(* IEC 61131-3 sources: ATCMcontrol_Engineering/src/Target/ATHW119/Libs/ATCM_System, 14 files *)

(* ---- _ThrowException.st ---- *)
(*[[
    UserURL= "ATCMfile:ThrowException.htm"
]]*)
(*
 *  ATCMControl Standard Function ThrowException
 *  Purpose: Throws an user exception for the calling task.
 *           NOTE: The task is stopped after the exception.
 *)
FUNCTION _ThrowException

inline{STDLIB(_ThrowException)}

END_FUNCTION

(* ---- ClearLocalTaskErrno.st ---- *)
(*[[
    UserURL= "ATCMfile:ClearLocalTaskErrno.htm"
]]*)
(*
 *  ATCMControl Standard Function ClearLocalTaskErrno
 *  Purpose: Clears the error state of the given task.
 *)
FUNCTION ClearLocalTaskErrno
VAR_INPUT
    NAME : ANY_STRING;
END_VAR

overload (STRING)  inline{STDLIB(ClearLocalTaskErrno)}

END_FUNCTION

(* ---- ClearTaskErrno.st ---- *)
(*[[
    UserURL= "ATCMfile:ClearTaskErrno.htm"
]]*)
(*
 *  ATCMControl Standard Function ClearTaskErrno
 *  Purpose: Clears the error state variable of the
 *           calling task. Error numbers <>0 signal an
 *           error.
 *)
FUNCTION ClearTaskErrno

inline{STDLIB(ClearTaskErrno)}

END_FUNCTION

(* ---- EnableWatchdog.st ---- *)
(*[[
    UserURL= "ATCMfile:EnableWatchdog.htm"
]]*)
(*
 *  ATCMControl Standard Function EnableWatchdog
 *)
FUNCTION EnableWatchdog

VAR_INPUT
    ENABLE : BOOL;
END_VAR

inline{STDLIB(EnableWatchdog)}

END_FUNCTION

(* ---- GetLocalTaskErrno.st ---- *)
(*[[
    UserURL= "ATCMfile:GetLocalTaskErrno.htm"
]]*)
(*
 *  ATCMControl Standard Function GetLocalTaskErrno
 *  Purpose: get the task error number of the named task.
 *           NOTE: name must be given in "lower case".
 *           Return values <>0 signal an error.
 *           See also the FC_ERRNO_* values
 *           defined in ATCM_System.cst.
 *)
FUNCTION GetLocalTaskErrno : DINT
VAR_INPUT
    NAME : ANY_STRING;
END_VAR

overload DINT(STRING)  inline {STDLIB(GetLocalTaskErrno)}

END_FUNCTION

(* ---- GetLocalTaskInfo.st ---- *)
(*[[
    UserURL= "ATCMfile:GetLocalTaskInfo.htm"
]]*)
(*
 *  ATCMControl Standard Function GetLocalTaskInfo
 *)
FUNCTION GetLocalTaskInfo
VAR_INPUT
    NAME : ANY_STRING;
END_VAR

VAR_IN_OUT
    INFO : TASKINFO;
END_VAR

overload (STRING,TASKINFO)  inline{STDLIB(GetLocalTaskInfo)}

END_FUNCTION

(* ---- GetLocalTaskState.st ---- *)
(*[[
    UserURL= "ATCMfile:GetLocalTaskState.htm"
]]*)
(*
 *  ATCMControl Standard Function GetLocalTaskState
 *  Purpose: get the current task execution state of the named task.
 *           NOTE: name must be given in "lower case".
 *  possible return values are (see system.cst):
 * CONST
 *   FC_TASK_STATE_ERROR       : DINT :=-1;
 *   FC_TASK_STATE_ONCREATION  : DINT := 0;
 *   FC_TASK_STATE_STOPPED     : DINT := 1;
 *   FC_TASK_STATE_RUNNING     : DINT := 2;
 *   FC_TASK_STATE_BREAK       : DINT := 3;
 * END_CONST
 *)
FUNCTION GetLocalTaskState : DINT
VAR_INPUT
    NAME : ANY_STRING;
END_VAR

overload DINT(STRING)  inline{STDLIB(GetLocalTaskState)}

END_FUNCTION

(* ---- GetTaskErrno.st ---- *)
(*[[
    UserURL= "ATCMfile:GetTaskErrno.htm"
]]*)
(*
 *  ATCMControl Standard Function GetTaskErrno
 *  Purpose: returns the last error number of the
 *           calling task.
 *           Return values <>0 signal an error.
 *           See also the FC_ERRNO_* values
 *           defined in ATCM_System.cst.
 *)
FUNCTION GetTaskErrno : DINT

inline{STDLIB(GetTaskErrno)}

END_FUNCTION

(* ---- getTimeSinceSystemBoot.st ---- *)
(*[[
    UserURL= "ATCMfile:getTimeSinceSystemBoot.htm"
]]*)

FUNCTION getTimeSinceSystemBoot : TIME

inline{STDLIB(GetTimeSinceSystemBoot)}

END_FUNCTION

(* ---- OutputDebugString.st ---- *)
(*[[
    UserURL= "ATCMfile:OutputDebugString.htm"
]]*)
(*
 *  ATCMControl Standard Functionblock OutputDebugString
 *  Purpose: Write a string to the control's standard output
 *           and the log file. A new line character is added
 *           automatically.
 *)
FUNCTION OutputDebugString
VAR_INPUT
    STR        : ANY_STRING;     (* a one-line message to the user*)
END_VAR

overload (STRING) inline{STDLIB(OutputDebugString)}

END_FUNCTION

(* ---- SFCResetToInitialStep.st ---- *)
(*[[
    UserURL= "ATCMfile:SFCResetToInitialStep.htm"
]]*)
(*
 *  ATCMControl Standard Function SFCResetToInitialStep
 *  Purpose: reset SFC logic
 *)
FUNCTION SFCResetToInitialStep

VAR_INPUT
    ENABLE : BOOL; (* reset only if ENABLE = TRUE *)
END_VAR

inline
{
    push1     %1
    POPD_IN_1    __resetSFC
}

END_FUNCTION

(* ---- StartLocalTask.st ---- *)
(*[[
    UserURL= "ATCMfile:StartLocalTask.htm"
]]*)
(*
 *  ATCMControl Standard Function StartLocalTask
 *  Purpose: Put the named task to the running state.
 *           NOTE: name must be given in "lower case".
 *)
FUNCTION StartLocalTask
VAR_INPUT
    NAME : ANY_STRING;
END_VAR

overload (STRING)  inline{STDLIB(StartLocalTask)}

END_FUNCTION

(* ---- StopLocalTask.st ---- *)
(*[[
    UserURL= "ATCMfile:StopLocalTask.htm"
]]*)
(*
 *  ATCMControl Standard Function StopLocalTask
 *  Purpose: Put the named task to the stopped state.
 *           NOTE: name must be given in "lower case".
 *  WARNING: never try to stop the own task.
 *)
FUNCTION StopLocalTask
VAR_INPUT
    NAME : ANY_STRING;
END_VAR

overload (STRING)  inline{STDLIB(StopLocalTask)}

END_FUNCTION

(* ---- SignalError.st ---- *)
(*[[
    UserURL= "ATCMfile:SignalError.htm"
]]*)
(*
 *  ATCMControl Standard Functionblock SignalError
 *  Purpose: Send Task to Error State
 *
 *  if enable=TRUE and errno<>0 then
 *    the current task is stopped.
 *)
FUNCTION_BLOCK SignalError

VAR_INPUT
    ENABLE     : BOOL:=TRUE;  (* enable this inst *)
    ERRNO      : DINT:=0;     (* error number *)
END_VAR

inline{STDLIB(SignalError)}

END_FUNCTION_BLOCK
